INTERFACE I_ValueDeviation

{attribute 'monitoring':='call'}
// Gets or sets the activation delay, before the deviation error is activated
PROPERTY ActivationDelay : TIME
GET
END_GET
SET
END_SET
END_PROPERTY

{attribute 'monitoring':='call'}
PROPERTY Enable : BOOL
GET
END_GET
SET
END_SET
END_PROPERTY

{attribute 'monitoring':='call'}
PROPERTY MaxDeviation : REAL
GET
END_GET
SET
END_SET
END_PROPERTY

{attribute 'monitoring':='call'}
PROPERTY Status : E_ValueDeviationStatus
GET
END_GET
END_PROPERTY

{attribute 'monitoring':='call'}
PROPERTY Value : REFERENCE TO ST_Value
GET
END_GET
END_PROPERTY

END_INTERFACE

(* stored: Version 1.1.0.1, ProductVersion 3.1.4024.13
   Itf I_ValueDeviation: Id {6463dd3b-c143-04a9-046e-1f54f26dd07e}
   Property ActivationDelay: Id {d7b8afe2-79da-0db0-2547-fe148212b733}
   Get Get: Id {4bd4909b-74da-0fc9-07c1-421fcf563df9}
   Set Set: Id {12d29bb2-fa0b-0b6c-0492-b1a210860132}
   Property Enable: Id {83252782-045e-0998-14c2-90c15608096c}
   Get Get: Id {dc2e45d2-94a1-034e-03ae-523883297a23}
   Set Set: Id {4711b673-5cf4-0c5e-1734-1dbc1399a762}
   Property MaxDeviation: Id {63135562-8145-0fb1-1b56-169d6afbfc32}
   Get Get: Id {92f3e69b-4296-091d-2944-efc94d8060a0}
   Set Set: Id {5855c4f4-48da-070c-1d8e-e0bb01c50e4b}
   Property Status: Id {a35f0f41-18e5-059d-06d8-1387bbebeda2}
   Get Get: Id {6918312a-ea4d-02bc-0604-db1166820882}
   Property Value: Id {2f10f158-c2f0-0478-00dc-74bb903b919b}
   Get Get: Id {142535be-b5ee-0119-2897-e80c20c729c4} *)
